# B&R Automation Studio project tcpip
Automation Studio 6.7.0.187

## Configuration SimAnsic

CPU , AutomationRuntime 6.7.6, Build 11.3.0

### Task classes (Cpu.sw)
```
Cyclic#2:
  tcp <- ANSIC.tcp.prg (BuildOptions=-W 6424)
  udp <- ANSIC.udp.prg
Binaries: arconfig, asfw, ashwd, iomap, sysconf
Libraries: AsArCfg, AsTcp, Operator, AsUdp, AsBrStr, brsystem, runtime, AsIecCon, astime
```

### Hardware
```
PLC1 : PC_any v1.1.2.0 (OrderNumber=PC)
  Connector IF1:
    ActivateIna = 1
  Connector IF2:
    ActivateIna = 1
  ConfigurationID = tcpip_Simulation
  XLinkUseDefault = 0
  FileDevice1
  FileDeviceName1 = USER
  FileDevicePath1 = USER_PATH
  ActivateWebServer = 0
  ActivateSdm = 0
  ActivateFtpServer = 1
```

## Configuration SimST

CPU , AutomationRuntime 6.7.6, Build 11.3.0, Safety 0.0

### Task classes (Cpu.sw)
```
Cyclic#2:
  tcp <- StructuredText.tcp.prg
  udp <- StructuredText.udp.prg
Binaries: arconfig, asfw, ashwd, iomap, sysconf
Libraries: AsArCfg, AsTcp, Operator, AsUdp, AsBrStr
```

### Hardware
same as Physical/SimAnsic/Hardware.hw

- Physical/SimST/PLC1/Cpu.per: same as Physical/SimAnsic/PLC1/Cpu.per
- Physical/SimST/PLC1/IoMap.iom: same as Physical/SimAnsic/PLC1/IoMap.iom
- Physical/SimST/PLC1/PvMap.vvm: same as Physical/SimAnsic/PLC1/PvMap.vvm
## Logical view

Binary libraries used (declarations not repeated): Operator, AsTcp, AsArCfg, AsUdp, brsystem, AsBrStr, Runtime, AsIecCon, astime

### Package Logical/ANSIC - Package

### Program Logical/ANSIC/tcp (ANSIC)

#### tcp.typ
```iecst
TYPE
	CLIENT_typ : 	STRUCT
		connected : BOOL;
		data_received : BOOL;
		addr : STRING[19];
		portclnt : UINT;
		receive_buffer : ARRAY[0..255]OF USINT;
		recv : TcpRecv;
		send : TcpSend;
		close : TcpClose;
	END_STRUCT;
	TcpSteps_enum :
		(
		SERVER_OPEN,
		SERVER_RUNNING,
		SERVER_ERROR
		);
END_TYPE
```

#### tcp.var
```iecst
VAR CONSTANT
	MAX_CLIENTS : USINT := 10;
	MAX_CLIENT_INDEX : USINT := MAX_CLIENTS-1;
END_VAR
VAR
	close : {REDUND_UNREPLICABLE} TcpClose;
	open : {REDUND_UNREPLICABLE} TcpOpen;
	server : {REDUND_UNREPLICABLE} TcpServer;
END_VAR
VAR CONSTANT
	PORT : UINT := 8000;
END_VAR
VAR
	step : {REDUND_UNREPLICABLE} TcpSteps_enum;
	step_str : {REDUND_UNREPLICABLE} STRING[79];
	client : {REDUND_UNREPLICABLE} ARRAY[0..MAX_CLIENT_INDEX] OF CLIENT_typ;
	tempstring : {REDUND_UNREPLICABLE} STRING[79];
	getipaddr : {REDUND_UNREPLICABLE} CfgGetIPAddr;
	myip : {REDUND_UNREPLICABLE} STRING[15];
	errstring : {REDUND_UNREPLICABLE} STRING[127];
	error : {REDUND_UNREPLICABLE} UINT;
	welcome_message : REFERENCE TO USINT;
	first_message : REFERENCE TO USINT;
	second_message : REFERENCE TO USINT;
END_VAR
```

#### tcp.c
```c
/* https://github.com/hilch/demo-AsTcp-AsUdp */

/* ------------------------------------------------------------------------------------------------------------
example for AsTCP- library
connect with 'tcpclient.py'. Multiple connections in parallel are possible.
---------------------------------------------------------------------------------------------------------------*/

#ifdef _DEFAULT_INCLUDES
#include <AsDefault.h>
#endif
#include <bur/plctypes.h>

char*				p_step_str;
char*				p_step_str_old;

/* --------------------------------------------------------------------------------------------------------
	startup after powerfail
--------------------------------------------------------------------------------------------------------
*/

void _INIT Initialisierung( void ){

	/* this could be useful when task is overloaded... */
	brsmemset( (UDINT) &open, 0, sizeof(open) );
	brsmemset( (UDINT) &close, 0, sizeof(close) );
	brsmemset( (UDINT) &server, 0, sizeof(server) );
	brsmemset( (UDINT) &getipaddr, 0, sizeof(getipaddr) );

	brsmemset( (UDINT) &client, 0, sizeof(client) );

	welcome_message = (USINT*) "Welcome to B&R Automation Runtime\nPress\n'1' for first message\n'2' for second message\n'3' to abort connection\n";
	first_message = (USINT*) "Hi Mickey Mouse\n";
	second_message = (USINT*) "Hi Donald Duck\n";

	server.enable = 1;

	getipaddr.enable = 1;
	getipaddr.pDevice = (UDINT) "IF2";
	getipaddr.pIPAddr = (UDINT) myip;
	getipaddr.Len = sizeof(myip);

	step = SERVER_OPEN;
	p_step_str = "INIT_UP";
	p_step_str_old = 0;
}

/* --------------------------------------------------------------------------------------------------------
	cyclic code
--------------------------------------------------------------------------------------------------------
*/

void _CYCLIC Zyklisch( void ){
	int i;

	CfgGetIPAddr( &getipaddr );
	if( getipaddr.status == 0 ){
		getipaddr.enable = 0;
	}

	switch( step ){
	case SERVER_OPEN:
		p_step_str = "TcpOpen()";
		open.enable = 1;
		open.pIfAddr = 0;
		open.port = PORT;
		open.options = tcpOPT_REUSEADDR ;
		TcpOpen( &open );
		if( open.status == 0 ){
			server.ident = open.ident;
			server.backlog = 10;
			server.pIpAddr = (UDINT) tempstring;
			step = SERVER_RUNNING;
		}
		else if( open.status != ERR_FUB_BUSY ){
			brsstrcpy( (UDINT) errstring, (UDINT) "error TcpOpen()" );
			error = open.status;
			step = SERVER_ERROR;
		}
		break;

	case SERVER_RUNNING:
		p_step_str = "server is running";
		TcpServer( &server );
		if( server.status == 0 ){  /* a new client has connected */
			for( i = 0; i < MAX_CLIENTS; ++i ){
				if( !client[i].connected ){
					client[i].connected = 1;
					brsstrcpy( (UDINT) client[i].addr, (UDINT) tempstring );
					client[i].recv.ident = server.identclnt;
					client[i].portclnt = server.portclnt;
					client[i].recv.enable = 1;
					client[i].recv.pData = (UDINT) client[i].receive_buffer;
					client[i].recv.datamax = sizeof(client[i].receive_buffer);
					client[i].recv.flags = 0;
					client[i].send.ident = server.identclnt;
					client[i].send.pData = (UDINT) welcome_message;
					client[i].send.datalen = brsstrlen( (UDINT) welcome_message );
					client[i].send.enable = 1;
					client[i].close.enable = 0;
					client[i].close.ident = server.identclnt;
					break;
				}
			}
		}

		/* Noodle through all clients */
		for( i = 0; i < MAX_CLIENTS; ++i ){

			/* receive data... */
			TcpRecv( &client[i].recv );

			if( client[i].recv.status == tcpERR_NOT_CONNECTED || client[i].recv.status == tcpERR_INVALID_IDENT || client[i].recv.status == tcpERR_SYSTEM ){
				client[i].close.enable = 1;
			}
			else if( client[i].recv.status == 0 ){
				if( client[i].recv.recvlen != 0 ){
					client[i].data_received = 1; /* Flag: Data has been received */
                }
                else if( client[i].recv.recvlen == 0 ){  /* Remote station has closed write direction */
                    client[i].close.enable = 1;
                }

			}

			/* Process input data ...*/
			if( client[i].data_received && client[i].send.enable == 0 ){  /* Data has arrived and send buffer is free */
				client[i].data_received = 0;
				switch( client[i].receive_buffer[0] ){
				case '1':
					client[i].send.pData = (UDINT) first_message;
					client[i].send.datalen = brsstrlen( (UDINT) client[i].send.pData );
					client[i].send.enable = 1;
					break;

				case '2':
					client[i].send.pData = (UDINT) second_message;
					client[i].send.datalen = brsstrlen( (UDINT) client[i].send.pData );
					client[i].send.enable = 1;
					break;

				case '3':
                    client[i].send.pData = (UDINT) "bye, bye\n";
                    client[i].send.datalen = brsstrlen( (UDINT) client[i].send.pData );
                    client[i].send.enable = 1;
					client[i].close.enable = 1;
					break;
				}
			}

			/* send output data */
			TcpSend( &client[i].send );
			if( client[i].send.status == 0 ){ /* sent successfully */
				client[i].send.enable = 0;
			}
			else if( (client[i].send.status != ERR_FUB_BUSY) && (client[i].send.status != ERR_FUB_ENABLE_FALSE) ){ /* error */
				client[i].send.enable = 0;
			}

			/* Release socket when connection is lost */
			TcpClose( &client[i].close );
            if( client[i].close.enable == 1 && client[i].close.status == 0 ){
               brsmemset( (UDINT) &client[i], 0, sizeof(CLIENT_typ) );
            }
		} /* end for( i = 0; i < MAX_CLIENTS... */

		break;

	case SERVER_ERROR:
		p_step_str = "error";

		break;

	}

	if( p_step_str != p_step_str_old ){
		p_step_str_old = p_step_str;
		brsstrcpy( (UDINT) step_str, (UDINT) p_step_str );
	}

}

/* --------------------------------------------------------------------------------------------------------
	is called on overload of the task
--------------------------------------------------------------------------------------------------------
*/

void _EXIT Exit( void ){
	int i;

	for( i = 0; i < MAX_CLIENTS; ++i ){
		do
			TcpClose( &client[i].close );
		while( client[i].close.status == ERR_FUB_BUSY );
	}

	do {
		close.enable = 1;
		close.ident = open.ident;
		close.how = 0;
		TcpClose( &close );
	}
	while( close.status == ERR_FUB_BUSY );

}
```

### Program Logical/ANSIC/udp (ANSIC)

#### udp.var - Local variables
```iecst
VAR CONSTANT
	PORT : UINT := 5000;
END_VAR
VAR
	sender_ip_addr : STRING[20];
	send_buffer : ARRAY[0..255] OF USINT;
	close : UdpClose;
	open : UdpOpen;
	send : UdpSend;
	receive_buffer : ARRAY[0..255] OF USINT;
	recv : UdpRecv;
END_VAR
```

#### udp.c - Implementation code
```c
/* https://github.com/hilch/demo-AsTcp-AsUdp */

/* ------------------------------------------------------------------------------------------------------------
example for AsTCP- library
connect with 'udpclient.py'.
---------------------------------------------------------------------------------------------------------------*/

#include <bur/plctypes.h>

#ifdef _DEFAULT_INCLUDES
 #include <AsDefault.h>
#endif

/* --------------------------------------------------------------------------------------------------------
   startup after powerfail
--------------------------------------------------------------------------------------------------------
*/

void _INIT Initialisierung( void )
{
    brsmemset( (UDINT) &open, 0, sizeof(open) );
    brsmemset( (UDINT) &close, 0, sizeof(close) );
    brsmemset( (UDINT) &recv, 0, sizeof(recv) );
    brsmemset( (UDINT) &send, 0, sizeof(send) );

    open.enable = 1;
	open.options = 0;//udpOPT_REUSEPORT;
    open.port = PORT;  /* receive port */
    open.pIfAddr = 0;
    UdpOpen( &open );

    recv.enable = 1;
    recv.ident = open.ident;
    recv.pData = (UDINT) &receive_buffer;
	recv.pIpAddr = (UDINT) sender_ip_addr;
    recv.datamax = sizeof(receive_buffer);

    send.enable = 1;
    send.ident = open.ident;
    send.flags = 0;
    send.pData = (UDINT) send_buffer;
    send.datalen = 0;

}

/* --------------------------------------------------------------------------------------------------------
    cyclic code
--------------------------------------------------------------------------------------------------------
*/

void _CYCLIC Zyklisch( void )
{
	UdpRecv( &recv );

	if( recv.status == 0 ){
		brsstrcpy( (UDINT) send_buffer, (UDINT) "echo: " );
		brsstrcat( (UDINT) send_buffer, (UDINT) receive_buffer );
		brsmemset( (UDINT) receive_buffer, 0 , sizeof(receive_buffer) );
		send.datalen = brsstrlen( (UDINT) send_buffer );
		send.pHost = (UDINT) sender_ip_addr; /* return back to sender */
		send.port = recv.port;
		send.enable = 1;
	}

    UdpSend( &send );
    if( send.enable && send.status != ERR_FUB_BUSY ){
        send.enable = 0;
		brsmemset( (UDINT) send_buffer, 0 , sizeof(send_buffer) );
    }

}

/* --------------------------------------------------------------------------------------------------------
   is called when overloading the task
--------------------------------------------------------------------------------------------------------
*/

void _EXIT Exit( void ){
    close.enable = 1;
    close.ident = open.ident;
    do {
        UdpClose( &close );
    }
    while( close.status == 65535 );

}
```


### Package Logical/StructuredText - Structured Text

### Program Logical/StructuredText/tcp (IEC) - Programm

#### tcp.typ
```iecst
TYPE
	TcpSteps_enum :
		(
		SERVER_OPEN,
		SERVER_RUNNING,
		SERVER_ERROR
		);
	CLIENT_typ : {REDUND_UNREPLICABLE} 	STRUCT
		connected : {REDUND_UNREPLICABLE} BOOL;
		data_received : {REDUND_UNREPLICABLE} BOOL;
		addr : {REDUND_UNREPLICABLE} STRING[19];
		portclnt : {REDUND_UNREPLICABLE} UINT;
		receive_buffer : {REDUND_UNREPLICABLE} ARRAY[0..255]OF USINT;
		recv : {REDUND_UNREPLICABLE} TcpRecv;
		send : {REDUND_UNREPLICABLE} TcpSend;
		close : {REDUND_UNREPLICABLE} TcpClose;
	END_STRUCT;
END_TYPE
```

#### tcp.var
```iecst
VAR
	i : {REDUND_UNREPLICABLE} DINT;
END_VAR
VAR CONSTANT
	PORT : UINT := 8000;
	MAX_CLIENTS : USINT := 10;
	MAX_CLIENT_INDEX : USINT := MAX_CLIENTS-1;
END_VAR
VAR
	close : {REDUND_UNREPLICABLE} TcpClose;
	open : {REDUND_UNREPLICABLE} TcpOpen;
	server : {REDUND_UNREPLICABLE} TcpServer;
	step : {REDUND_UNREPLICABLE} TcpSteps_enum;
	step_str : {REDUND_UNREPLICABLE} STRING[79] := '';
	client : {REDUND_UNREPLICABLE} ARRAY[0..MAX_CLIENT_INDEX] OF CLIENT_typ;
	tempstring : {REDUND_UNREPLICABLE} STRING[79] := '';
	getipaddr : {REDUND_UNREPLICABLE} CfgGetIPAddr;
	myip : {REDUND_UNREPLICABLE} STRING[15];
	errstring : {REDUND_UNREPLICABLE} STRING[127];
	error : {REDUND_UNREPLICABLE} UINT;
END_VAR
VAR CONSTANT
	welcome_message : STRING[128] := 'Welcome TO B&R Automation Runtime$nPress$n$'1$' for first message$n$'2$' for second message$n$'3$' TO abort connection$n';
	first_message : STRING[128] := 'Hi Mickey Mouse$n';
	second_message : STRING[128] := 'Hi Donald Duck$n';
END_VAR
```

#### tcp.st - Implementierungscode
```iecst
(* https://github.com/hilch/demo-AsTcp-AsUdp *)

(*
example FOR AsTCP- library
connect with 'tcpclient.py'. Multiple connections in parallel are possible.
*)

(* startup after powerfail *)
PROGRAM _INIT

	(* this could be useful when task is overloaded... *)
	brsmemset( ADR(open), 0, SIZEOF(open) );
	brsmemset( ADR(close), 0, SIZEOF(close) );
	brsmemset( ADR(server), 0, SIZEOF(server) );
	brsmemset( ADR(getipaddr), 0, SIZEOF(getipaddr) );

	brsmemset( ADR(client), 0, SIZEOF(client) );

	server.enable := 1;

	getipaddr.enable := 1;
	getipaddr.pDevice := ADR('IF2');
	getipaddr.pIPAddr := ADR(myip);
	getipaddr.Len := SIZEOF(myip);

	step := SERVER_OPEN;

END_PROGRAM

(* cyclic code *)
PROGRAM _CYCLIC

	getipaddr();
	IF getipaddr.status = 0 THEN
		getipaddr.enable := FALSE;
	END_IF

	CASE step OF
	SERVER_OPEN:
		step_str := 'TcpOpen()';
		open.enable := TRUE;
		open.pIfAddr := 0;
		open.port := PORT;
		open.options := tcpOPT_REUSEADDR ;
		open();
		IF open.status = 0 THEN
			server.ident := open.ident;
			server.backlog := 10;
			server.pIpAddr := ADR(tempstring);
			step := SERVER_RUNNING;
		ELSIF open.status <> ERR_FUB_BUSY THEN
			errstring := 'error TcpOpen()';
			error := open.status;
			step := SERVER_ERROR;
		END_IF

	SERVER_RUNNING:
		step_str := 'server is running';
		server();
		IF  server.status = 0 THEN  (* a new client has connected *)
			FOR i := 0 TO (MAX_CLIENTS-1) DO
				IF NOT(client[i].connected)THEN
					client[i].connected := TRUE;
					client[i].addr := tempstring;
					client[i].recv.ident := server.identclnt;
					client[i].portclnt := server.portclnt;
					client[i].recv.enable := TRUE;
					client[i].recv.pData := ADR(client[i].receive_buffer);
					client[i].recv.datamax := SIZEOF(client[i].receive_buffer);
					client[i].recv.flags := 0;
					client[i].send.ident := server.identclnt;
					client[i].send.pData := ADR(welcome_message);
					client[i].send.datalen := brsstrlen(ADR(welcome_message));
					client[i].send.enable := TRUE;
					client[i].close.enable := FALSE;
					client[i].close.ident := server.identclnt;
					EXIT;
				END_IF
			END_FOR
		END_IF

		(* Noodle through all clients *)
		FOR i := 0 TO (MAX_CLIENTS-1) DO
			(* receive data... *)
			client[i].recv();

			IF client[i].recv.status = tcpERR_NOT_CONNECTED OR client[i].recv.status = tcpERR_INVALID_IDENT OR client[i].recv.status = tcpERR_SYSTEM THEN
				client[i].close.enable := TRUE;
			ELSIF client[i].recv.status = 0 THEN
				IF client[i].recv.recvlen <> 0 THEN
					client[i].data_received := TRUE; (* Flag: Data has been received *)
				ELSIF client[i].recv.recvlen = 0 THEN  (* Remote station has closed write direction *)
					client[i].close.enable := TRUE;
				END_IF
            END_IF

			(* Process input data ...*)
			IF client[i].data_received AND client[i].send.enable = 0 THEN  (* Data has arrived AND send buffer is free *)
				client[i].data_received := FALSE;
				CASE client[i].receive_buffer[0] OF
					49:  (* ascii '1' *)
					client[i].send.pData := ADR(first_message);
					client[i].send.datalen := brsstrlen( client[i].send.pData );
					client[i].send.enable := TRUE;

					50: (* ascii '2' *)
					client[i].send.pData := ADR(second_message);
					client[i].send.datalen := brsstrlen( client[i].send.pData );
					client[i].send.enable := TRUE;

					51: (* ascii '3' *)
					client[i].send.pData := ADR('bye, bye$n');
					client[i].send.datalen := brsstrlen( client[i].send.pData );
					client[i].send.enable := TRUE;
					client[i].close.enable := TRUE;
				END_CASE
			END_IF

			(* send output data *)
			client[i].send();
			IF client[i].send.status = 0 THEN (* sent successfully *)
				client[i].send.enable := FALSE;
			ELSIF client[i].send.status <> ERR_FUB_BUSY AND client[i].send.status <> ERR_FUB_ENABLE_FALSE THEN (* error *)
				client[i].send.enable := FALSE;
			END_IF

			(* Release socket when connection is lost *)
			client[i].close();
			IF client[i].close.enable AND client[i].close.status = 0 THEN
				brsmemset( ADR(client[i]), 0, SIZEOF(CLIENT_typ) );
			END_IF
		END_FOR

	SERVER_ERROR:
		step_str := 'error';

	END_CASE

END_PROGRAM

(* is called on overload of the task *)
PROGRAM _EXIT

	FOR i := 0 TO (MAX_CLIENTS-1) DO
		REPEAT
			client[i].close();
			UNTIL client[i].close.status <> ERR_FUB_BUSY
		END_REPEAT
	END_FOR

	REPEAT
		close.enable := TRUE;
		close.ident := open.ident;
		close.how := 0;
		close();
		UNTIL close.status <> ERR_FUB_BUSY
	END_REPEAT

END_PROGRAM
```

### Program Logical/StructuredText/udp (IEC)

#### udp.var - Local variables
```iecst
VAR CONSTANT
	PORT : UINT := 5000;
END_VAR
VAR
	sender_ip_addr : STRING[20];
	send_buffer : ARRAY[0..255] OF USINT;
	close : UdpClose;
	open : UdpOpen;
	send : UdpSend;
	receive_buffer : ARRAY[0..255] OF USINT;
	recv : UdpRecv;
END_VAR
```

#### udp.st - Implementation code
```iecst
(* https://github.com/hilch/demo-AsTcp-AsUdp *)

(* --------------------------------------------------------------------------------------------------------
   startup after powerfail
--------------------------------------------------------------------------------------------------------
*)

PROGRAM _INIT

    brsmemset( ADR(open), 0, SIZEOF(open) );
    brsmemset( ADR(close), 0, SIZEOF(close) );
    brsmemset( ADR(recv), 0, SIZEOF(recv) );
    brsmemset( ADR(send), 0, SIZEOF(send) );

    open.enable := TRUE;
	open.options := 0; //udpOPT_REUSEPORT;
    open.port := PORT;  (* receive port *)
    open.pIfAddr := 0;
    open();

    recv.enable := TRUE;
    recv.ident := open.ident;
    recv.pData := ADR(receive_buffer);
	recv.pIpAddr := ADR(sender_ip_addr);
    recv.datamax := SIZEOF(receive_buffer);

    send.enable := TRUE;
    send.ident := open.ident;
    send.flags := 0;
    send.pData := ADR(send_buffer);
    send.datalen := 0;

END_PROGRAM

(* --------------------------------------------------------------------------------------------------------
    cyclic code
--------------------------------------------------------------------------------------------------------
*)

PROGRAM _CYCLIC

	recv();

	IF recv.status = 0 THEN
		brsstrcpy( ADR(send_buffer), ADR('echo:') );
		brsstrcat( ADR(send_buffer), ADR(receive_buffer) );
		brsmemset( ADR(receive_buffer), 0 , SIZEOF(receive_buffer) );
		send.datalen := brsstrlen( ADR(send_buffer) );
		send.pHost := ADR(sender_ip_addr); (* return back to sender *)
		send.port := recv.port;
		send.enable := TRUE;
	END_IF

    send();

    IF send.enable AND send.status <> ERR_FUB_BUSY THEN
        send.enable := FALSE;
		brsmemset( ADR(send_buffer), 0 , SIZEOF(send_buffer) );
    END_IF

END_PROGRAM

(* --------------------------------------------------------------------------------------------------------
   is called when overloading the task
--------------------------------------------------------------------------------------------------------
*)

PROGRAM _EXIT

    close.enable := TRUE;
    close.ident := open.ident;
    REPEAT
        close();
    	UNTIL close.status <> ERR_FUB_BUSY
    END_REPEAT

END_PROGRAM
```
